PROGRAM startup_sequence
VAR
END_VAR

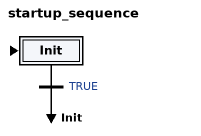
INITIAL_STEP Init:
END_STEP
TRANSITION FROM Init TO Init
    := TRUE;
END_TRANSITION

END_PROGRAM

(* stored: Version 1.1.0.1, ProductVersion 3.1.4024.13
   POU startup_sequence: Id {0e3660d3-54c7-4e4c-988c-e32bb4d8d93c}, SpecialFunc None *)
